Fanuc KAREL source: CA0061.KL

PROGRAM CA0061
%STACKSIZE=65535
%PRIORITY=65535
%NOLOCKGROUP
TYPE
T=STRUCTURE
A : INTEGER
B : REAL
ENDSTRUCTURE
VAR
G : INTEGER
I : INTEGER
R : REAL
B : BOOLEAN
S : STRING[16]
AI : ARRAY[2] OF INTEGER
AR : ARRAY[2] OF REAL
ST : T
P : XYZWPR
V : VECTOR
ROUTINE F(P1 : INTEGER; P2 : INTEGER; P3 : INTEGER; P4 : INTEGER; P5 : INTEGER; P6 : INTEGER; P7 : INTEGER; P8 : INTEGER) FROM CA0061
ROUTINE F
BEGIN
G=(G + 1)
END F
BEGIN
G=0
I=1
R=2.5
B=TRUE
S='A'
AI[1]=3
AR[1]=4.5
-- UNSAFE_SOURCE_IR line 38: ST.A = 5
-- UNSAFE_SOURCE_IR line 39: ST.B = 6.5
-- UNSAFE_SOURCE_IR line 40: F(I, ARG_2_UNRESOLVED, I, ARG_4_UNRESOLVED, I, ARG_6_UNRESOLVED, I, ARG_8_UNRESOLVED)
END CA0061
